  def pop_up_config_g_et_d():
      close_popup()
      popup3 = "popup CONFIGURATION : Les deux tables sont configurées."
      socket_open("127.0.0.1",29999,"internal") # open internal socket
      socket_send_line(popup3,"internal")     #Affichage message
      socket_send_byte(10,"internal")
  end

  def pop_up_config_g():
      close_popup()
      popup3 = "popup CONFIGURATION : Table droite configurée."
      socket_open("127.0.0.1",29999,"internal") # open internal socket
      socket_send_line(popup3,"internal")     #Affichage message
      socket_send_byte(10,"internal")
  end
  $ 53 "Mouvements soudures"
  $ 54 "Script: fcts_balayage.script"
  def fct_determineAxeBalayage(p_start,p_stop):

      global  diff_x = norm(p_start[0]-p_stop[0])
      global  diff_y = norm(p_start[1]-p_stop[1])
      global  diff_z = norm(p_start[2]-p_stop[2])

      global offset_x =  0
      global offset_y =  0
      global offset_z = 0

      local tolerance = 0.02



      if ( (diff_z >0.05) ):
          offset_z = 1
      end

      if ( (diff_x >tolerance) or (offset_z == 1)):
          offset_y = 1
      end

      if ( (diff_y >tolerance) or (offset_z == 1)):
          offset_x = 1
      end

  end

  def fct_set_offset():

      if (offset_x == 1):
          offset[0] = sin((i/cycle_duration)*2.0*pi) * amplitude
      end

      if (offset_y == 1):
          offset[1] = sin((i/cycle_duration)*2.0*pi) * amplitude
      end

  end

  thread runBalayage():
    while (True):
        global ctrl_frequency=350.0
        global weave_frequency=1.2
        global amplitude=0.003
        global cycle_duration=(ctrl_frequency / weave_frequency)
        global pi=3.14159
        global offset=[0.0, 0.0, 0.0, 0.0, 0.0, 0.0]
        global i=0
        path_offset_enable()
        global alpha=0.1
        path_offset_set_alpha_filter(alpha)

        while (True):
          fct_set_offset()
          path_offset_set(offset, 2)
          global i=i+1
          sync()
        end
      end

  end

  def fct_activerBalayage(p_start, p_stop):

      fct_determineAxeBalayage(p_start,p_stop)
      global thr_runBalayage = run runBalayage()

  end

  def fct_desactiverBalayage():

      kill thr_runBalayage

  end
  $ 55 "Script: fcts_ralentir_fin_ligne.script"
  def fct_calcul_point_inter(p_debut,p_fin):

      local p_inter = p_fin

      local poucentage = 0.95
      local inc = 0
      local vecteur_global = p[0,0,0,0,0,0]
      local vecteur_reduit = p[0,0,0,0,0,0]

      while (inc < 6):   #a valider avec d'autres tests (peut etre faire une moyenne)
          vecteur_global[inc] = p_fin[inc] - p_debut[inc]
          vecteur_reduit[inc] = vecteur_global[inc]*poucentage
          p_inter[inc] = p_debut[inc] + vecteur_reduit[inc]
          inc = inc +1
      end

      return p_inter
    end


  $ 56 "General"
  $ 57 "Script: diverses.script"
  def attente_carters_ouverts():
      # vérifier que les carter sont ouverts,
      # sinon attendre en faisant clignoter les leds

      while ((get_configurable_digital_in(add_SecuGaucheOk) == True) or (get_configurable_digital_in(add_SecuDroiteOK) == True)):

          sync()
          # 94 "'clingottement pour signifier qu'il y  un defaut sur un des carters '"
          set_standard_digital_out(add_Dcy_Voyant, False)
          set_configurable_digital_out(add_Led_Arret, False)
          sleep(0.5)
          set_standard_digital_out(add_Dcy_Voyant, True)
          set_configurable_digital_out(add_Led_Arret, True)
          sleep(0.5)
          sync()
      end

      #carter OK, RAZ des sorties
      set_standard_digital_out(add_Dcy_Voyant, False)
      set_configurable_digital_out(add_Led_Arret, False)
      sleep(2)
      sync()

  end

  def deplacement_depart_init():

      global angle_base = get_actual_joint_positions ()
      if (angle_base[0] <= 0.7):
          if (angle_base[0] >= 1.6):
              # 116 "Départ"        A CHANGER PAR UNE POSTION ENREGISTREE
              movej(pose_depart, a = accelerationHorsSoudure, v = vitesseHorsSoudure)
          else:
              if (angle_base[0] > 1.6):
                  movej(Point_init_D, a = accelerationHorsSoudure, v = vitesseHorsSoudure)
                  movej(Point_avt_initD, a = accelerationHorsSoudure, v = vitesseHorsSoudure)
              else:
                  if (angle_base[0] < 0.7):
                      movej(Point_init_G, a = accelerationHorsSoudure, v = vitesseHorsSoudure)
                  end
              end
          end
      else:
          # 124 "SinonSi angle_base[0]>1.6"
          if (angle_base[0] > 1.6):

              movej(Point_init_D, a = accelerationHorsSoudure, v = vitesseHorsSoudure)
              movej(Point_avt_initD, a = accelerationHorsSoudure, v = vitesseHorsSoudure)
          else:
              if (angle_base[0] < 0.7):
                  movej(Point_init_G, a = accelerationHorsSoudure, v = vitesseHorsSoudure)
              end
          end
      end
      # 131 "Départ"             A CHANGER PAR UNE POSTION ENREGISTREE
      movej(pose_depart, a = accelerationHorsSoudure, v = vitesseHorsSoudure)
      #global angle_base= get_actual_joint_positions ()
      sync()
  end





  def mode_configuration():
      #nouveau

      if ((config_g == 1) and (config_d == 1)):
          pop_up_config_g_et_d()
      elif ((config_g == 1) and (config_d == 0)):
          pop_up_config_g()
      elif ((config_g == 0) and (config_d == 1)):
          pop_up_config_d()
      elif ((config_g == 0) and (config_d == 0)):
          pop_up_config()
      end

      while ((get_configurable_digital_in(add_ModeManu) == False  ) and (get_standard_digital_in(add_bp_ConfigReglage) == False  )):
          thread Thread_while_145():
              while (True):  # faire clignoter les voyants des tables, pour informer de l'attente d'une action
                  set_standard_digital_out(add_VoyantTableDroite, True)
                  set_standard_digital_out(add_VoyantTableGauche, False)
                  sleep(0.5)
                  set_standard_digital_out(add_VoyantTableDroite, False)
                  set_standard_digital_out(add_VoyantTableGauche, True)
                  sleep(0.5)
                  sync()
              end
          end
          if (get_standard_digital_in(adresse_bp_d) == False and get_standard_digital_in(adresse_bp_g) == False and get_configurable_digital_in(add_ModeManu) == False and get_standard_digital_in(add_bp_ConfigReglage) == False):
              global thread_handler_145 = run Thread_while_145()
              while (get_standard_digital_in(adresse_bp_d) == False and get_standard_digital_in(adresse_bp_g) == False and get_configurable_digital_in(add_ModeManu) == False and get_standard_digital_in(add_bp_ConfigReglage) == False):
                  sync()
              end
              kill thread_handler_145
          end
          if (get_standard_digital_in(adresse_bp_g) == True): #table gauche
              set_standard_digital_out(add_VoyantTableGauche, True)
              set_standard_digital_out(add_VoyantTableDroite, False)
              movej(Point_init_G, a = accelerationHorsSoudure, v = vitesseHorsSoudure, r = 0.006)
              movej(Point_Attente_G, a = accelerationHorsSoudure, v = vitesseHorsSoudure, r = 0.006)
              movej(Point_config_g, a = accelerationHorsSoudure, v = vitesseHorsSoudure)
              global led_cobot = 1
              fun_config_g()
              global led_cobot = 0
              fun_valid_config_g()
              movej(Point_Attente_G, a = accelerationHorsSoudure, v = vitesseHorsSoudure, r = 0.006)
              movej(Point_init_G, a = accelerationHorsSoudure, v = vitesseHorsSoudure, r = 0.006)
              # 170 "Départ"         A CHANGER PAR UNE POSTION ENREGISTREE
              movej(pose_depart, a = accelerationHorsSoudure, v = vitesseHorsSoudure)
          end

          if (get_standard_digital_in(adresse_bp_d) == True): #table droite
              set_standard_digital_out(add_VoyantTableDroite, True)
              set_standard_digital_out(add_VoyantTableGauche, False)
              movej(Point_avt_initD, a = accelerationHorsSoudure, v = vitesseHorsSoudure, r = 0.006)
              movej(Point_init_D, a = accelerationHorsSoudure, v = vitesseHorsSoudure)
              movej(Point_Attente_D, a = accelerationHorsSoudure, v = vitesseHorsSoudure, r = 0.006)
              movej(Point_config_d, a = accelerationHorsSoudure, v = vitesseHorsSoudure)
              global led_cobot = 1
              fun_config_d()
              global led_cobot = 0
              fun_valid_config_d()
              movej(Point_Attente_D, a = accelerationHorsSoudure, v = vitesseHorsSoudure, r = 0.006)
              movej(Point_init_D, a = accelerationHorsSoudure, v = vitesseHorsSoudure, r = 0.006)
              movej(Point_avt_initD, a = accelerationHorsSoudure, v = vitesseHorsSoudure, r = 0.006)
              # 190 "Départ"         A CHANGER PAR UNE POSTION ENREGISTREE
              movej(pose_depart, a = accelerationHorsSoudure, v = vitesseHorsSoudure)
          end
      end

      sync()
  end




  def mode_Reglage():
      #Pas à Pas
      if ((config_g == 1) and (config_d == 1)):
          pop_up_reg_gd()
          global boucle = 1
      elif ((config_g == 1) and (config_d == 0)):
          pop_up_reg_gd()
          global boucle = 1
      elif ((config_g == 0) and (config_d == 1)):
          pop_up_reg_d()
          global boucle = 1
      else:
          close_popup()
          while (get_standard_digital_in(add_bp_ConfigReglage) == True):
              popup("Aucune configuration n'est actuellement detectée.", "Erreur", False, True, blocking = True)
          end
      end
  end

  end
  global boucle = 1
  while ((get_configurable_digital_in(add_ModeManu) == False  ) and (boucle == 1) and (get_standard_digital_in(add_bp_ConfigReglage) == True  )):
      thread Thread_while_208():
          while (True):
              if (config_g == 1):
                  set_standard_digital_out(add_VoyantTableGauche, True)
              end
              if (config_d == 1):
                  set_standard_digital_out(add_VoyantTableDroite, True)
              end
              sleep(0.5)
              set_standard_digital_out(add_VoyantTableGauche, False)
              set_standard_digital_out(add_VoyantTableDroite, False)
              sleep(0.5)
          end
      end
      if (get_standard_digital_in(adresse_bp_d) == False and get_standard_digital_in(adresse_bp_g) == False and get_configurable_digital_in(add_ModeManu) == False and get_standard_digital_in(add_bp_ConfigReglage) == True):
          global thread_handler_208 = run Thread_while_208()
          while (get_standard_digital_in(adresse_bp_d) == False and get_standard_digital_in(adresse_bp_g) == False and get_configurable_digital_in(add_ModeManu) == False and get_standard_digital_in(add_bp_ConfigReglage) == True):
              sync()
          end
          kill thread_handler_208
      end
      if (get_standard_digital_in(adresse_bp_g) == True): #table gauche
          global safe_mode = 1
          set_standard_digital_out(add_VoyantTableGauche, True)
          set_standard_digital_out(add_VoyantTableDroite, False)
          movej(Point_init_G, a = accelerationHorsSoudure, v = vitesseHorsSoudure, r = 0.006)
          movej(Point_Attente_G, a = accelerationHorsSoudure, v = vitesseHorsSoudure, r = 0.006)
          movej(pose_inter_g, a = accelerationHorsSoudure, v = vitesseHorsSoudure)
          global led_cobot = 1
          fun_Pas_A_Pas_g()
          global led_cobot = 0
          global safe_mode = 0
          global boucle = 0
      end
      if (get_standard_digital_in(adresse_bp_d) == True): #table droite
          global safe_mode = 1
          set_standard_digital_out(add_VoyantTableDroite, True)
          set_standard_digital_out(add_VoyantTableGauche, False)
          movej(Point_avt_initD, a = accelerationHorsSoudure, v = vitesseHorsSoudure, r = 0.006)
          movej(Point_init_D, a = accelerationHorsSoudure, v = vitesseHorsSoudure, r = 0.006)
          movej(pose_inter_d, a = accelerationHorsSoudure, v = vitesseHorsSoudure)
          global led_cobot = 1
          fun_Pas_A_Pas_d()
          global led_cobot = 0
          global safe_mode = 0
          global boucle = 0
      end
  end

  sync()
  end

  def mode_Execution():

      if ((config_g == 1) and (config_d == 1)):
          pop_up_exe()
          global boucle = 1
      elif ((config_g == 1) and (config_d == 0)):
          pop_up_exe_g()
          global boucle = 1
      elif ((config_g == 0) and (config_d == 1)):
          pop_up_exe_d()
          global boucle = 1
      else:
          close_popup()
          while (get_configurable_digital_in(add_ModeManu) == True):
              popup("Aucune programmation n'est actuellement detectée, veillez à programmer une pièce avant de vouloir l'éxécuter.", "Erreur", False, True, blocking = True)
          end
      end

      while (( get_configurable_digital_in(add_ModeManu) == True  ) and (boucle == 1)):
          thread Thread_while_259():
              while (True):
                  if (config_g == 1):
                      set_standard_digital_out(add_VoyantTableGauche, True)
                  end
                  if (config_d == 1):
                      set_standard_digital_out(add_VoyantTableDroite, True)
                  end
                  sleep(0.5)
                  set_standard_digital_out(add_VoyantTableGauche, False)
                  set_standard_digital_out(add_VoyantTableDroite, False)
                  sleep(0.5)
              end
          end
          if (get_standard_digital_in(adresse_bp_d) == False and get_standard_digital_in(adresse_bp_g) == False and get_configurable_digital_in(add_ModeManu) == True):
              global thread_handler_259 = run Thread_while_259()
              while (get_standard_digital_in(adresse_bp_d) == False and get_standard_digital_in(adresse_bp_g) == False and get_configurable_digital_in(add_ModeManu) == True):
                  sync()
              end
              kill thread_handler_259
          end
          if ((get_standard_digital_in(adresse_bp_g) == True  ) and (config_g == True  )):
              global boucle_g = 1
              while (boucle_g == 1):
                  set_configurable_digital_out(add_CmdCarterBit1, True)
                  set_standard_digital_out(add_VoyantTableGauche, True)
                  set_standard_digital_out(add_VoyantTableDroite, False)
                  sleep(0.25)
                  set_standard_digital_out(add_VoyantTableGauche, False)
                  sleep(0.25)
                  if (get_configurable_digital_in(add_SecuGaucheOk) == False):
                      set_standard_digital_out(add_VoyantTableGauche, True)
                      if (get_configurable_digital_in(add_SecuGaucheOk) == False):
                          close_popup()
                          while (get_configurable_digital_in(add_SecuGaucheOk) == False):
                              sync()
                          end
                      end
                  end
                  if (get_configurable_digital_in(add_SecuGaucheOk) == True):
                      global secu_g = 1
                      set_standard_digital_out(add_VoyantTableGauche, True)
                      movej(Point_init_G, a = accelerationHorsSoudure, v = vitesseHorsSoudure, r = 0.006)
                      fun_execution_g()
                      movej(Point_Attente_G, a = accelerationHorsSoudure, v = vitesseHorsSoudure, r = 0.006)
                      movej(Point_init_G, a = accelerationHorsSoudure, v = vitesseHorsSoudure, r = 0.006)
                      # 294 "Départ"         A CHANGER PAR UNE POSTION ENREGISTREE
                      movej(pose_depart, a = accelerationHorsSoudure, v = vitesseHorsSoudure)
                      set_configurable_digital_out(add_CmdCarterBit1, False)
                      global secu_g = 0
                      global boucle_g = 0
                  end
              end
              global boucle = 0
          else:
              if ((get_standard_digital_in(adresse_bp_g) == True  ) and (config_g == False  )):
                  close_popup()
                  popup("Aucune programmation n'est actuellement detectée sur la table gauche, veillez à programmer une pièce avant de vouloir l'éxécuter.", "Erreur", False, True, blocking = True)
                  global boucle = 0
              end
          end
          if ((get_standard_digital_in(adresse_bp_d) == True  ) and (config_d == True  )):
              global boucle_d = 1
              pop_up_deb_exe_d()
              while (boucle_d == 1):
                  set_configurable_digital_out(add_CmdCarterBit2, True)
                  set_standard_digital_out(add_VoyantTableGauche, False)
                  set_standard_digital_out(add_VoyantTableDroite, True)
                  sleep(0.25)
                  set_standard_digital_out(add_VoyantTableDroite, False)
                  sleep(0.25)
                  if (get_configurable_digital_in(add_SecuDroiteOK) == False):
                      set_standard_digital_out(add_VoyantTableDroite, True)
                      sleep(6.0)
                      if (get_configurable_digital_in(add_SecuDroiteOK) == False):
                          close_popup()
                          while (get_configurable_digital_in(add_SecuDroiteOK) == False):
                              sync()
                          end
                      end
                  end
                  if (get_configurable_digital_in(add_SecuDroiteOK) == True):
                      global secu_d = 1
                      set_standard_digital_out(add_VoyantTableDroite, True)
                      movej(Point_avt_initD, a = accelerationHorsSoudure, v = vitesseHorsSoudure)
                      fun_execution_d()
                      set_configurable_digital_out(add_CmdCarterBit2, False)
                      global secu_d = 0
                      global boucle_d = 0
                  end
              end
              global boucle = 0
          else:
              if ((get_standard_digital_in(adresse_bp_d) == True  ) and (config_d == False  )):
                  close_popup()
                  popup("Aucune programmation n'est actuellement detectée sur la table droite, veillez à programmer une pièce avant de vouloir l'éxécuter.", "Erreur", False, True, blocking = True)
                  global boucle = 0
              end
          end
      end
      sync()
  end
  $ 58 "Script: general2.script"
  def General():

      while (True):

          #INTIALISATION
          safe_mode = 0
          set_configurable_digital_out(add_CmdCarterBit1, False) #stop commande carter
          set_configurable_digital_out(add_CmdCarterBit2, False)

          attente_carters_ouverts() #éviter un contact avec le bras
          # LIGNE 23 GENERAL

          deplacement_depart_init() #premier déplacement à gérer en focntion de la position réel du robot lors de l'init
          #LIGNE 54 GENERAL

          # TEST DES MODES :

          # lecture de la postion des Bps
          if ((get_configurable_digital_in(add_ModeManu) == False) and (get_standard_digital_in(add_bp_ConfigReglage) == False)):
              mode_configuration()#l 55-> 127
          elif ((get_configurable_digital_in(add_ModeManu) == False) and (get_standard_digital_in(add_bp_ConfigReglage) == True  )):
              mode_Reglage() #l 127 -> 199
          elif (get_configurable_digital_in(add_ModeManu) == True):
              mode_Execution() #
          else:
              #faire erreur
          end
      end



  end
  $ 72 "Thread_1"
  thread Thread_1():
    while (True):
      $ 73 "Test_Ordre_Marche"
      $ 74 "If Test_Ordre_Mar≟ True "
      if (Test_Ordre_Mar ==   True  ):
        $ 75 "If config_d ≟ 1  or  config_g ≟ 1"
        if (config_d  ==  1   or   config_g  ==  1):
          $ 76 "Set Ordre_Marche=On"
          set_standard_digital_out(0, True)
          $ 77 "Wait: 0.5"
          sleep(0.5)
          $ 78 "If Reponse_Ordre≟ False "
          if (get_standard_digital_in(4) ==   False  ):
            $ 79 "'Si aucune reponse n'a etait recue, arret du programme'"
            # 'Si aucune reponse n'a etait recue, arret du programme'
            $ 80 "close_popup()"
            close_popup()
            $ 81 "Popup: Defaut : L'Ordre marche a ete coupe ( le poste est peu-etre eteint ) "
            popup("Defaut : L'Ordre marche a ete coupe ( le poste est peu-etre eteint ) ", "Error", False, True, blocking=False)
            halt
          end
          $ 82 "Test_Ordre_Mar≔ False "
          global Test_Ordre_Mar=  False
          $ 83 "sync()"
          sync()
        end
      end
      $ 84 "Erreur ordre marche pendant utilisation"
      $ 85 "If Arc_On≟ True   and Reponse_Arc≟ True  and Reponse_Ordre≟ False "
      if (get_standard_digital_out(1) ==   True     and  get_standard_digital_in(5) ==   True    and  get_standard_digital_in(4) ==   False  ):
        $ 86 "'Test pour savoir si ordre marche a ete coupe pendant utilisation'"
        # 'Test pour savoir si ordre marche a ete coupe pendant utilisation'
        $ 87 "close_popup()"
        close_popup()
        $ 88 "Popup: Defaut : Mise sous puissance coupee pendant la trajectoire"
        popup("Defaut : Mise sous puissance coupee pendant la trajectoire", "Error", False, True, blocking=False)
        halt
      end
      $ 89 "sync()"
      sync()
    end
  end
  threadId_Thread_1 = run Thread_1()
  $ 90 "Thread_2"
  thread Thread_2():
    while (True):
      $ 91 "mode_soudure"
      $ 92 "If Mode_soudure ≟  True "
      if (get_configurable_digital_in(3)  ==    True  ):
        $ 93 "If Mode_soudure≟ True  and soudure_on ≟ True "
        if (get_configurable_digital_in(3) ==   True    and  soudure_on  ==   True  ):
          $ 94 "fin_soud≔0"
          global fin_soud=0
          $ 95 "Test_Ordre_Mar≔ True "
          global Test_Ordre_Mar=  True
          $ 96 "Test_Job≔ True "
          global Test_Job=  True
          $ 97 "Wait Test_Ordre_Mar≟ False "
          while (not(Test_Ordre_Mar ==   False  )):
            sync()
          end
          $ 98 "Wait Test_Job≟ False "
          while (not(Test_Job ==   False  )):
            sync()
          end
          $ 99 "Set Arc_On=On"
          set_standard_digital_out(1, True)
          $ 100 "Test_Gaz≔ True "
          global Test_Gaz=  True
          $ 101 "'Test_Gaz permet de faire un appel dans le thread pour tester l'arriver gaz'"
          # 'Test_Gaz permet de faire un appel dans le thread pour tester l'arriver gaz'
          $ 102 "Wait Valide_Gaz≟ True "
          while (not(Valide_Gaz ==   True  )):
            sync()
          end
          $ 103 "'Valide_Gaz permet  de connaitre quand le traitement de l'arriver gaz est terminer ans le thread.'"
          # 'Valide_Gaz permet  de connaitre quand le traitement de l'arriver gaz est terminer ans le thread.'
        else:
          $ 104 "ElseIf Mode_soudure ≟ True  and soudure_on ≟ False "
          if (get_configurable_digital_in(3)  ==   True    and  soudure_on  ==   False  ):
            $ 105 "'Attente post debit gaz'"
            # 'Attente post debit gaz'
            $ 106 "Set Arc_On=Off"
            set_standard_digital_out(1, False)
            $ 107 "Test_Gaz≔ False "
            global Test_Gaz=  False
            $ 108 "Loop Reponse_Arc ≟ 1"
            while (get_standard_digital_in(5)  ==  1):
              $ 109 "fin_soud≔0"
              global fin_soud=0
              $ 110 "sync()"
              sync()
            end
            $ 111 "fin_soud≔1"
            global fin_soud=1
          end
        end
      end
      $ 112 "sync()"
      sync()
    end
  end
  threadId_Thread_2 = run Thread_2()
  $ 113 "Thread_3"
  thread Thread_3():
    while (True):
      $ 114 "led_cobot_2"
      $ 115 "If led_cobot ≟ True "
      if (led_cobot  ==   True  ):
        $ 116 "If valider_bp_co ≟ True "
        if (get_tool_digital_in(0)  ==   True  ):
          $ 117 "Set TO[1]=On"
          set_tool_digital_out(1, True)
          $ 118 "Wait: 0.25"
          sleep(0.25)
          $ 119 "Set TO[1]=Off"
          set_tool_digital_out(1, False)
          $ 120 "Wait: 0.25"
          sleep(0.25)
          $ 121 "Set TO[1]=On"
          set_tool_digital_out(1, True)
          $ 122 "Wait: 0.25"
          sleep(0.25)
          $ 123 "Set TO[1]=Off"
          set_tool_digital_out(1, False)
          $ 124 "Wait: 0.25"
          sleep(0.25)
          $ 125 "Set TO[1]=On"
          set_tool_digital_out(1, True)
          $ 126 "Wait: 0.25"
          sleep(0.25)
          $ 127 "Set TO[1]=Off"
          set_tool_digital_out(1, False)
          $ 128 "Wait: 0.25"
          sleep(0.25)
          $ 129 "sync()"
          sync()
        end
        $ 130 "sync()"
        sync()
      end
      $ 131 "sync()"
      sync()
      $ 132 "sync()"
      sync()
    end
  end
  threadId_Thread_3 = run Thread_3()
  $ 133 "Thread_4"
  thread Thread_4():
    while (True):
      $ 134 "led_cobot"
      $ 135 "If led_cobot ≟ True "
      if (led_cobot  ==   True  ):
        $ 136 "Loop led_cobot ≟  True "
        while (led_cobot  ==    True  ):
          $ 137 "Set TO[0]=On"
          set_tool_digital_out(0, True)
          $ 138 "Wait: 0.5"
          sleep(0.5)
          $ 139 "Set TO[0]=Off"
          set_tool_digital_out(0, False)
          $ 140 "Wait: 0.5"
          sleep(0.5)
          $ 141 "sync()"
          sync()
        end
        $ 142 "sync()"
        sync()
      else:
        $ 143 "Else" "noBreak"
        $ 144 "Set TO[0]=Off"
        set_tool_digital_out(0, False)
        $ 145 "Set TO[1]=Off"
        set_tool_digital_out(1, False)
      end
      $ 146 "sync()"
      sync()
    end
  end
  threadId_Thread_4 = run Thread_4()
  $ 147 "Thread_5"
  thread Thread_5():
    while (True):
      $ 148 "Test_Arc_On"
      $ 149 "Erreur gaz pendant utilisation"
      $ 150 "Timer_gaz"
      $ 151 "If Test_Gaz≟ True "
      if (Test_Gaz ==   True  ):
        $ 152 "Wait: 1.0"
        sleep(1.0)
        $ 153 "Loop Reponse_Arc≟ False  and Arc_On≟ True "
        thread Thread_while_153():
          while (True):
            $ 154 "'La boucle permet d'activer le timer et tester deux condition pour les Defaults'"
            # 'La boucle permet d'activer le timer et tester deux condition pour les Defaults'
            $ 155 "timer_ret_gaz: Start"
            timer_ret_gaz_is_counting = True
            $ 156 "If timer_ret_gaz>0.5"
            global thread_flag_156=0
            thread Thread_if_156():
              $ 157 "'Le timer permet de realiser une attente '"
              # 'Le timer permet de realiser une attente '
              $ 158 "close_popup()"
              close_popup()
              $ 159 "Popup: Defaut : Pas de retour flux, stabilisation gaz"
              popup("Defaut : Pas de retour flux, stabilisation gaz", "Error", False, True, blocking=False)
              halt
              thread_flag_156 = 1
            end
            if (timer_ret_gaz>0.5):
              global thread_handler_156=run Thread_if_156()
              while (thread_flag_156 == 0):
                if not(timer_ret_gaz>0.5):
                  kill thread_handler_156
                  thread_flag_156 = 2
                else:
                  sync()
                end
              end
            else:
              thread_flag_156 = 2
            end
            if (thread_flag_156 == 2):
              $ 160 "ElseIf Reponse_Ordre≟ False "
              if (get_standard_digital_in(4) ==   False  ):
                $ 161 "'Cette condition nous permet de pouvoir tout couper ordre marche pendant la boucle.'"
                # 'Cette condition nous permet de pouvoir tout couper ordre marche pendant la boucle.'
                $ 162 "close_popup()"
                close_popup()
                $ 163 "Popup: Defaut : Perte retour de signal, mise sous puissance generateur"
                popup("Defaut : Perte retour de signal, mise sous puissance generateur", "Error", False, True, blocking=False)
                halt
              end
            end
          end
        end
        if (get_standard_digital_in(5) ==   False    and  get_standard_digital_out(1) ==   True  ):
          global thread_handler_153=run Thread_while_153()
          while (get_standard_digital_in(5) ==   False    and  get_standard_digital_out(1) ==   True  ):
            sync()
          end
          kill thread_handler_153
        end
        $ 164 "Valide_Gaz≔ True "
        global Valide_Gaz=  True
        $ 165 "timer_ret_gaz: Reset"
        timer_ret_gaz = 0
      end
      $ 166 "sync()"
      sync()
    end
  end
  threadId_Thread_5 = run Thread_5()
  $ 167 "Thread_6"
  thread Thread_6():
    while (True):
      $ 168 "Test_Job"
      $ 169 "If Test_Job≟ True "
      if (Test_Job ==   True  ):
        $ 173 "Test_Job≔ False "
        global Test_Job=  False
      end
      $ 174 "sync()"
      sync()
    end
  end
  threadId_Thread_6 = run Thread_6()
  $ 175 "Thread_7"
  thread Thread_7():
    while (True):
      $ 176 "secu"
      $ 177 "If SecuGaucheOk ≟  False  and secu_g ≟ 1"
      if (get_configurable_digital_in(4)  ==    False    and  secu_g  ==  1):
        $ 178 "close_popup()"
        close_popup()
        $ 179 "Popup: ATTENTION : Defaut carter !"
        popup("ATTENTION : Defaut carter !", "Error", False, True, blocking=False)
        halt
      else:
        $ 180 "ElseIf SecuDroiteOk ≟ False  and secu_d ≟ 1"
        if (get_configurable_digital_in(5)  ==   False    and  secu_d  ==  1):
          $ 181 "close_popup()"
          close_popup()
          $ 182 "Popup: ATTENTION : Defaut carter !"
          popup("ATTENTION : Defaut carter !", "Error", False, True, blocking=False)
          halt
        end
      end
      $ 183 "sync()"
      sync()
    end
  end
  threadId_Thread_7 = run Thread_7()
  $ 184 "Thread_8"
  thread Thread_8():
    while (True):
      $ 185 "bloq_soud_arret"
      $ 186 "If Mode_soudure≟ False  and Test_Gaz ≟ True "
      if (get_configurable_digital_in(3) ==   False    and  Test_Gaz  ==   True  ):
        $ 187 "close_popup()"
        close_popup()
        $ 188 "Popup: Defaut : L'ordre de soudure a ete coupe pendant l'utilisation."
        popup("Defaut : L'ordre de soudure a ete coupe pendant l'utilisation.", "Error", False, True, blocking=False)
        halt
      end
      $ 195 "sync()"
      sync()
    end
  end
  threadId_Thread_8 = run Thread_8()
  $ 206 "Thread_10"
  thread Thread_10():
    while (True):
      $ 207 "reglage"
      $ 208 "If safe_mode ≟ 1  and Mode_manu ≟  True "
      if (safe_mode  ==  1   and  get_configurable_digital_in(7)  ==    True  ):
        $ 209 "close_popup()"
        close_popup()
        $ 210 "Popup: STOP !!!!"
        popup("STOP !!!!", "Error", False, True, blocking=False)
        halt
      end
      $ 211 "sync()"
      sync()
      $ 212 "sync()"
      sync()
    end
  end
  threadId_Thread_10 = run Thread_10()
  $ 59 "Robot Program"
  $ 61 "General()"
  General()
end
